Staubli VAL3: JointAccel.dtx

public num ja[6]
